Universal Robots PolyScope program: ControlSet5.urp

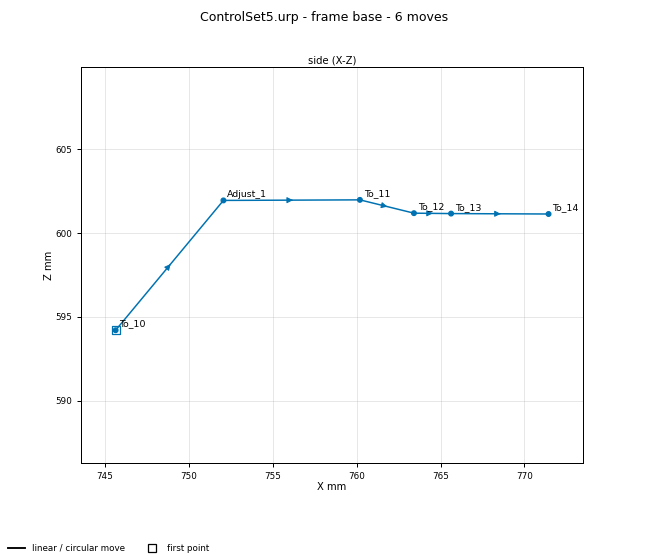
[picture p0: tool path of ControlSet5.urp in frame base, 6 of 8 moves have a stored position in this frame; points joined in program order, loops and branches not executed]
Program ControlSet5 (installation=Youssef directory=/programs/Youssef createdIn=5.9.5.1031259 lastSavedIn=5.9.5.1031259 robotSerialNumber=20215500597)
Calibrated DH parameters: a=[0.000193, -0.066673, -0.391568, -0.000012, 0.00005, 0]; d=[0.162643, -472.05677, 465.132521, 7.058239, 0.099746, 0.099582]; alpha=[1.571116, 0.00089, 0.003862, 1.569269, -1.569248, 0]; deltaTheta=[0, -1.413394, 7.628392, 0.068187, 0, -0.000001]
Robot Program (runOnlyOnce=true)
  MoveL speed 250 mm/s, acceleration 1200 mm/s^2 (useActiveTCP=true) feature=Base
    Waypoint Waypoint (Variable): variable(featureName=Control_Standby)
    Waypoint Waypoint (Variable): variable(featureName=Control_R_Strt)
    Waypoint To_10: TCP in base x=745.639 y=-17.849 z=594.209 mm, rx=-0.0636 ry=2.4703 rz=-0.2743 rad; joints [169.914, -71.977, 43.233, -100.537, -93.87, 75.587] deg; TCP offset x=0 y=0 z=191.5 mm, rx=0 ry=0 rz=0 rad
  MoveL speed 250 mm/s, acceleration 1200 mm/s^2 (useActiveTCP=true) feature=Base
    Waypoint Adjust_1: TCP in base x=752.062 y=-17.854 z=601.945 mm, rx=-0.0636 ry=2.4704 rz=-0.2743 rad; joints [170.031, -70.021, 39.176, -98.427, -93.941, 75.669] deg
    Waypoint To_11: TCP in base x=760.195 y=-17.853 z=601.978 mm, rx=-0.0636 ry=2.4703 rz=-0.2743 rad; joints [170.175, -68.462, 36.913, -97.718, -94.032, 75.776] deg
  MoveL speed 250 mm/s, acceleration 1200 mm/s^2 (useActiveTCP=true) feature=Base
    Waypoint To_12: TCP in base x=763.415 y=-17.79 z=601.185 mm, rx=-0.0639 ry=2.4729 rz=-0.2738 rad; joints [170.234, -67.759, 35.895, -97.252, -94.064, 75.817] deg
  MoveL speed 250 mm/s, acceleration 1200 mm/s^2 (useActiveTCP=true) feature=Base
    Waypoint To_13: TCP in base x=765.628 y=-17.8 z=601.16 mm, rx=-0.0639 ry=2.4729 rz=-0.2738 rad; joints [170.271, -67.314, 35.235, -97.032, -94.088, 75.845] deg
  MoveL speed 250 mm/s, acceleration 1200 mm/s^2 (useActiveTCP=true) feature=Base
    Waypoint To_14: TCP in base x=771.437 y=-17.779 z=601.135 mm, rx=-0.064 ry=2.473 rz=-0.2737 rad; joints [170.371, -66.115, 33.43, -96.418, -94.148, 75.918] deg
